// TIA Portal V20 export
FUNCTION_BLOCK "Lift_Drive_To_Level"   // FB7, LAD
{ S7_Optimized_Access := 'TRUE' }
// stored: MemoryReserve 100, SetENOAutomatically false
   VAR_INPUT
      QR_ReaderST34 : DInt;
      QR_ReaderST32 : DInt;
      Selected_Level : SInt;
      Drive_To_Pos : Bool;
   END_VAR
   VAR_OUTPUT
      Jog_Forward : Bool;
      Jog_Backward : Bool;
      Velocity : LReal;
      Lift_On_Floor_Number : SInt;
   END_VAR
   VAR
      Safe_Distance_QR1_QR2 { ExternalAccessible := 'False'; ExternalVisible := 'False'; ExternalWritable := 'False'} : Int := 150;
      Alarm : Byte;   // X0-Crossed platform,
      Dis_Level : Array[0..6] of DInt;
      ABS_Distance : LReal;
   END_VAR
   VAR CONSTANT
      Tolerance : SInt := 5;
      Nominal_Velocity : LReal := 1500.0;
      Slow_Down_Distance : LReal := 1000.0;
   END_VAR
BEGIN

REGION Network 1 (SCL): X0-Crossed platform,
   #Alarm.%X0 := (#QR_ReaderST32 - #QR_ReaderST34) >= #Safe_Distance_QR1_QR2;
END_REGION

REGION Network 2 (SCL): Drive to selected floor
   IF #Drive_To_Pos AND NOT #Alarm.%X0 THEN

       IF ABS(#QR_ReaderST32 - #Dis_Level[#Selected_Level]) <= #Tolerance THEN
           // in tolerance
           #Jog_Forward := FALSE;
           #Jog_Backward := FALSE;

       ELSIF #QR_ReaderST32 > #Dis_Level[#Selected_Level] THEN
           #Jog_Backward := TRUE;
           #Jog_Forward := FALSE;

       ELSE
           #Jog_Forward := TRUE;
           #Jog_Backward := FALSE;

       END_IF;
   END_IF;
END_REGION

REGION Network 3 (SCL): Set velocity
   #ABS_Distance := ABS(#QR_ReaderST32 - #Dis_Level[#Selected_Level]);

   IF #Drive_To_Pos AND NOT #Alarm.%X0 THEN

       IF #ABS_Distance <= #Tolerance THEN
           // in position
           #Velocity := 0.0;

       ELSIF #ABS_Distance >= #Slow_Down_Distance THEN
           // far position / max velocity
           #Velocity := #Nominal_Velocity;

       ELSE
           // breaking
           #Velocity := (#ABS_Distance / #Slow_Down_Distance) * #Nominal_Velocity;

           // minimum 5%
           IF #Velocity < (#Nominal_Velocity * 0.05) THEN
               #Velocity := #Nominal_Velocity * 0.05;
           END_IF;

       END_IF;

   END_IF;

   IF NOT #Drive_To_Pos AND NOT #Alarm.%X0 AND #ABS_Distance <= #Tolerance THEN
       #Lift_On_Floor_Number := #Selected_Level;
   END_IF;
END_REGION
END_FUNCTION_BLOCK
